PROGRAM MAIN
VAR
	starter	:	DigitalOutput;
	input	:	DigitalInput;
	output	:	DigitalOutput;
	term	:	DigitalInput;
	counter	:	UINT	:=	0;
	c_limit	:	UINT 	:= 100;
	s_limit	:	UINT	:=90;
	
END_VAR


IF counter < c_limit THEN
	counter := counter + 1;
ELSIF counter >= c_limit THEN
	counter := 0;
END_IF;

IF counter > s_limit THEN
	starter.out := 1;
ELSE
	starter.out := 0;
END_IF

IF input.in THEN
	output.out := 1;
ELSE
	output.out := 0;
END_IF

END_PROGRAM

(* stored: Version 1.1.0.1, ProductVersion 3.1.4020.12
   POU MAIN: Id {41f7eedd-d7ab-4487-8081-0ce2740c8596}, SpecialFunc None *)
